// TwinCAT 3 PLC project PlcIotMqttSampleAwsIoTButton
// ProgramVersion: 3.1.4021.2
// libraries:
//   Tc2_Standard, * (Beckhoff Automation GmbH)
//   Tc2_System, * (Beckhoff Automation GmbH)
//   Tc3_IotBase, * (Beckhoff Automation GmbH)
//   Tc3_JsonXml, * (Beckhoff Automation GmbH)
//   Tc3_Module, * (Beckhoff Automation GmbH)
// project tree:
//   DUTs/ ST_IotButton.TcDUT
//   / PlcTask.TcTTO
//   POUs/ MAIN.TcPOU (not stored), PrgMqttCom.TcPOU
// real-time tasks:
//   TASK PlcTask: cycle T#10ms, priority 20, ADS port 350

CONFIGURATION PlcIotMqttSampleAwsIoTButton
    RESOURCE PLC ON TwinCAT3
        TASK PlcTask(INTERVAL := T#10ms, PRIORITY := 20);
        PROGRAM MAIN WITH PlcTask : MAIN;
    END_RESOURCE
END_CONFIGURATION

// ---- DUTs/ST_IotButton.TcDUT
(* Possible payloads of Amazon IoT Button *)
(* {"serialNumber":"G030PT028191AC4R","batteryVoltage":"1547mV","clickType":"SINGLE"} *)
(* {"serialNumber":"G030PT028191AC4R","batteryVoltage":"1547mV","clickType":"DOUBLE"} *)
TYPE ST_IotButton :
STRUCT
	serialNumber 	: STRING(255);	// Serial number as shown on back of device
	batteryVoltage 	: STRING(255);	// [mv]
	clickType		: STRING(255);	// SINGLE, DOUBLE
	configuration	: STRING(255);	// Initial event after configuration  
END_STRUCT
END_TYPE

// ---- POUs/PrgMqttCom.TcPOU
PROGRAM PrgMqttCom
VAR
	fbMqttClient : FB_IotMqttClient;
	bSetParameter : BOOL := TRUE;
	bConnect : BOOL := TRUE;
	
	(* topic subscribtion *)
	bSubscribed : BOOL;
	sTopicSub : STRING(255) := 'iotbutton/G030PT028191AC4R';

	(* received message *)	
	{attribute 'TcEncoding':='UTF-8'}
	sTopicRcv : STRING(255);
	{attribute 'TcEncoding':='UTF-8'}
	sPayloadRcv : STRING(255);
	stIotButton : ST_IotButton;
	
	(* JSON *)
	fbJson 			: FB_JsonDomParser;
	jsonDoc 		: SJsonValue;
	jsonProp		: SJsonValue;
	jsonValue		: SJsonValue;
	jsonIt			: SJsonIterator;
	bHasMember		: BOOL;
	sm				: STRING;
	sj 				: SJsonValue;	
	
	fbMessageQueue : FB_IotMqttMessageQueue;
	fbMessage : FB_IotMqttMessage;
	
	hrErrorOccurred : HRESULT; // contains the latest occurred error
END_VAR

IF bSetParameter THEN
	bSetParameter := FALSE;
	
	(* TLS settings for AWS IoT connection *)
	fbMqttClient.stTLS.sCA := 'c:\TwinCAT\3.1\Config\Certificates\root.pem';
    fbMqttClient.stTLS.sCert := 'c:\TwinCAT\3.1\Config\Certificates\e4090580c5-certificate.pem.crt';
    fbMqttClient.stTLS.sKeyFile := 'c:\TwinCAT\3.1\Config\Certificates\e4090580c5-private.pem.key';
	
	(* Broker settings für AWS IoT *)
	fbMqttClient.sHostName:= 'a158o5z7vk6zkt.iot.us-west-2.amazonaws.com';
	fbMqttClient.nHostPort:= 8883;
	fbMqttClient.sClientId:= 'SVENG-NB04'; 

	fbMqttClient.ipMessageQueue := fbMessageQueue;
END_IF

fbMqttClient.Execute(bConnect);
IF fbMqttClient.bError THEN
	// add your error logging here
	hrErrorOccurred := fbMqttClient.hrErrorCode;
END_IF
IF fbMessageQueue.nQueuedMessages > 0 THEN
	IF fbMessageQueue.Dequeue(fbMessage:=fbMessage) THEN
		fbMessage.GetTopic(pTopic:=ADR(sTopicRcv), nTopicSize:=SIZEOF(sTopicRcv) );
		fbMessage.GetPayload(pPayload:=ADR(sPayloadRcv), nPayloadSize:=SIZEOF(sPayloadRcv), bSetNullTermination:=FALSE);

		(* Retrieve JSON content *)
		jsonDoc := fbJson.ParseDocument(sPayloadRcv);
		bHasMember := fbJson.HasMember(jsonDoc, 'serialNumber');
		IF (bHasMember) THEN
			bHasMember := FALSE;
	  		jsonProp := fbJson.FindMember(jsonDoc, 'serialNumber');
			stIotButton.serialNumber := fbJson.GetString(jsonProp);
	  	END_IF

		bHasMember := fbJson.HasMember(jsonDoc, 'batteryVoltage');
		IF (bHasMember) THEN
			bHasMember := FALSE;
	  		jsonProp := fbJson.FindMember(jsonDoc, 'batteryVoltage');
			stIotButton.batteryVoltage := fbJson.GetString(jsonProp);
	  	END_IF		

		bHasMember := fbJson.HasMember(jsonDoc, 'clickType');
		IF (bHasMember) THEN
			bHasMember := FALSE;
	  		jsonProp := fbJson.FindMember(jsonDoc, 'clickType');
			stIotButton.clickType := fbJson.GetString(jsonProp);
	  	END_IF			

		bHasMember := fbJson.HasMember(jsonDoc, 'configuration');
		IF (bHasMember) THEN
			bHasMember := FALSE;
	  		jsonProp := fbJson.FindMember(jsonDoc, 'configuration');
			stIotButton.configuration := fbJson.GetString(jsonProp);
	  	END_IF
	END_IF
END_IF

IF fbMqttClient.bConnected THEN
	IF NOT bSubscribed THEN
		bSubscribed := fbMqttClient.Subscribe(sTopic:=sTopicSub, eQoS:=TcIotMqttQos.AtMostOnceDelivery);
		IF fbMqttClient.bError THEN
			// add your error logging here
			hrErrorOccurred := fbMqttClient.hrErrorCode;
		END_IF
	END_IF
END_IF

END_PROGRAM
